# EPICS substitutions: apps/bcmApp/Db/bcm.substitutions
file "db/rate.template" {
pattern
 {P, C}
 {hc, 1}
 {hc, 2}
 {hc, 3}
 {hc, 4}
 {hc, 5}
 {hc, 6}
 {hc, 7}
 {hc, 8}
 {hc, 9}
 {hc, 10}
 {hc, 11}
 {hc, 12}
 {hc, 13}
 {hc, 14}
 {hc, 15}
 {hc, 16}
}
